// TIA Portal V19 export
// export: Created 2025-04-23T01:58:05.8009231Z, ExportSetting WithDefaults, DisplayName Totally Integrated Automation Portal, DisplayVersion V19, DisplayName TIA Portal Openness, DisplayVersion V19, DisplayName TIA Portal Version Control Interface, DisplayVersion V19, DisplayName STEP 7 Professional, DisplayVersion V19, DisplayName STEP 7 Safety, DisplayVersion V19, DisplayName WinCC Basic/Comfort/Advanced, DisplayVersion V19, DisplayName WinCC Unified, DisplayVersion V19
FUNCTION_BLOCK "Block_4"   // FB2, SCL
{ S7_Optimized_Access := 'TRUE' }
VERSION : 0.1
// stored: AutoNumber true, IsIECCheckEnabled false, IsRetainMemResEnabled false, MemoryReserve 100, SetENOAutomatically false, UDAEnableTagReadback false
   VAR_INPUT
      m1 : Int;
      m2 : Int;
   END_VAR
   VAR_OUTPUT
      m3 : Int;
   END_VAR
BEGIN
   #m3 := #m1 - #m2;
END_FUNCTION_BLOCK
